# EPICS autosave request: ADApp/Db/apex2_settings.req
$(P)$(R)ReadSFRMTimeout
$(P)$(R)NumDarks
